// TIA Portal V21 export
TYPE "Std_Zona"
   STRUCT
      In : Struct
         RichiestaLampadaReset : Bool;
      END_STRUCT;
      Gen : Struct   // Generale
         UpdatePrm_Mem : Bool;   // Memoria di update parametri
         UpdatePrm : Bool;   // Sistema e resetta memorie delle utenze e nella strumentazione
         ResetLoc_Hmi : Bool;   // Reset locale della zona da HMI
         Reset : Bool;   // Ingresso reset allarmi
      END_STRUCT;
      Prm : Struct
         CentralinaOkDaTempo { S7_SetPoint := 'True'} : "Std_stTimer";   // Centralina sicurezza ripristinata + tempo
         RitardoCicloAuto { S7_SetPoint := 'True'} : "Std_stTimer";   // Ritardo all'inserzione del ciclo automatico
         RitardoCicloMan { S7_SetPoint := 'True'} : "Std_stTimer";   // Ritardo all'inserzione del ciclo manuale
         RitardoStopDaTempo { S7_SetPoint := 'True'} : "Std_stTimer";
      END_STRUCT;
      Dati : Struct
         BloccoRichiamato : Bool;
      END_STRUCT;
      Allarmi : Struct
         Prm : Struct
            PulisciStoricoUtenze : Bool;   // Pulisci storico slot allarmi da utenze con pulsante di reset
         END_STRUCT;
         SlotAllarmeDaUtenze : Array[0.."K_NumSlotAllarmiDaUtenze"] of Struct   // Storico degli allarmi che si sono settati nella zona
            Allarme : Bool;   // Slot occupato da un allarme
            AllarmeSilenziato : Bool;   // L'allarme è stato silenziato
            TipoNum : Int;   // Tipologia di utenza in allarme scritto in numero
            TipoNome : String[10];   // Tipologia di utenza in allarme scritto in lettere
            Indice : Int;   // Numero dell'utenza nell'array
            NumAllarme : Int;
         END_STRUCT;
         "A" { S7_SetPoint := 'True'} : Array[0.."K_NumAllarmiPerZone"] of "Std_PrmAllarmeStd";   // Allarmi standard della zona
         AG { S7_SetPoint := 'True'} : Array[0..15] of "Std_PrmAllarmeStd";   // Allarmi generici specifici per ogni zona
         WordHMI { S7_SetPoint := 'True'} : Word;   // Word per lista segnalazioni HMI
         WordHMI_AG { S7_SetPoint := 'True'} : Word;   // Word per lista segnalazioni HMI
      END_STRUCT;
      Out : Struct   // Ciclo
         Auto : Bool;   // Ciclo automatico attivo
         Man : Bool;   // Ciclo manuale attivo
         Attivo : Bool;   // Almeno un ciclo attivo
         StopDaTempo : Bool;
         Attesa : Bool;
         AutoDaHmi : Bool;   // Tipo di ciclo richiesto ad HMI (1 = auto / 0 = man)
         Stato : Int;   // 0=CicloOf 1=CicloManOn 2=CicloAutoOn 3=Attesa 4=Segnalazione 5=Allarme
         CumulativoAllarmi : Bool;   // Almeno un allarme presente
         SirenaSuona : Bool;   // Richiesta di far suonare l'allarme
         CentralinaOk { S7_SetPoint := 'True'} : Bool;   // Centralina sicurezza ripristinata
      END_STRUCT;
      Rif_Inc : Struct
         K_Zona_Padre : Int;
      END_STRUCT;
   END_STRUCT;
   // Prm.CentralinaOkDaTempo.Preset := 1.0;
   // Prm.RitardoCicloAuto.Preset := 1.0;
   // Prm.RitardoCicloMan.Preset := 1.0;
   // // Allarmi."A"[1] : Centralina di sicurezza
   // // Allarmi."A"[2] : Ciclo non inserito
END_TYPE
